Universal Robots PolyScope program: washer_get_glass.urp

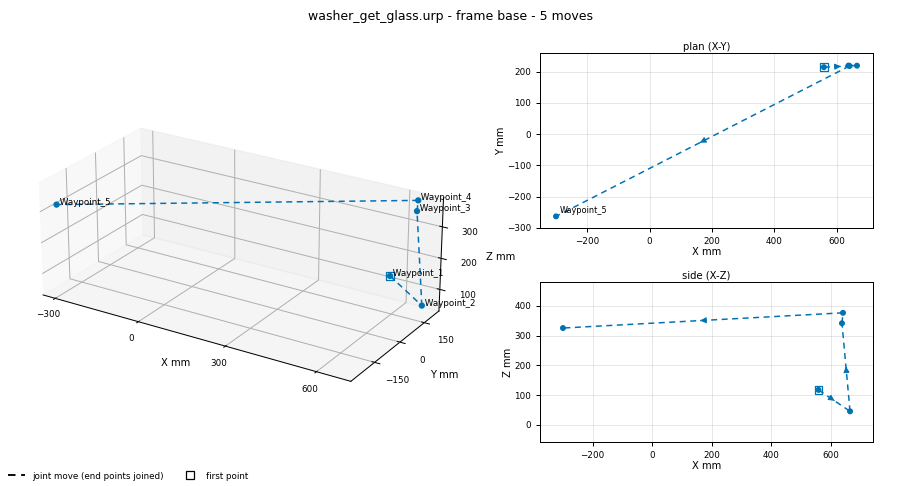
[picture p0: tool path of washer_get_glass.urp in frame base, 5 of 5 moves have a stored position in this frame; points joined in program order, loops and branches not executed]
Program washer_get_glass (installation=default directory=/programs createdIn=5.9.5.1031259 lastSavedIn=5.9.5.1031259 robotSerialNumber=20215500597)
Calibrated DH parameters: a=[0.000193, -0.066673, -0.391568, -0.000012, 0.00005, 0]; d=[0.162643, -472.05677, 465.132521, 7.058239, 0.099746, 0.099582]; alpha=[1.571116, 0.00089, 0.003862, 1.569269, -1.569248, 0]; deltaTheta=[0, -1.413394, 7.628392, 0.068187, 0, -0.000001]
Robot Program (runOnlyOnce=false)
  MoveJ speed 60 deg/s, acceleration 80 deg/s^2 (useActiveTCP=true) feature=Base
    Waypoint Waypoint_1: TCP in base x=558.375 y=214.785 z=117.374 mm, rx=-0.0094 ry=1.6112 rz=-0.0088 rad; joints [195.765, -72.945, 133.044, 302.22, 105.904, -90.017] deg; TCP offset x=0 y=0 z=191.5 mm, rx=0 ry=0 rz=0 rad
    URCap Gripper Activate (Robotiq_Grippers, Robotiq Inc.) dataModel(ResetAndActivateKey=true)
    URCap Gripper (Robotiq_Grippers, Robotiq Inc.) dataModel(position=0.0, force=40.0, speed=49.80392156862745, positionInDouble=0.0, forceInDouble=40.0, speedInDouble=49.80392156862745, slaveIds=[9], blocking=true)
    Waypoint Waypoint_2: TCP in base x=664.345 y=219.439 z=45.438 mm, rx=0.0376 ry=1.6347 rz=-0.0606 rad; joints [194.828, -54.791, 116.729, 301.842, 108.519, -89.734] deg
    URCap Gripper (Robotiq_Grippers, Robotiq Inc.) dataModel(position=90.19607843137254, force=50.0, speed=40.0, positionInDouble=90.19607843137254, forceInDouble=50.0, speedInDouble=40.0, slaveIds=[9], blocking=true)
    Waypoint Waypoint_3: TCP in base x=637.232 y=219.943 z=341.244 mm, rx=-0.0272 ry=1.665 rz=-0.0791 rad; joints [194.822, -85.852, 103.444, 347.962, 106.824, -92.22] deg
    Waypoint Waypoint_4: TCP in base x=640.64 y=218.481 z=376.237 mm, rx=2.2037 ry=-0.0464 rz=2.1952 rad; joints [194.824, -87.164, 103.426, 343.909, 107.316, -269.899] deg
    Waypoint Waypoint_5: TCP in base x=-299.672 y=-263.204 z=325.11 mm, rx=1.1501 ry=-1.1061 rz=1.2274 rad; joints [328.599, -97.097, 126.286, 342.336, -31.887, -282.051] deg
    Halt
